PROGRAM MAIN
VAR
END_VAR

END_PROGRAM

(* stored: Version 1.1.0.1
   POU MAIN: Id {5ba7a48c-9cd2-4db4-ab93-9c6b2a606dc4} *)
